(* PLC project  *)

CONFIGURATION Empty_Module_2
END_CONFIGURATION
